// SIMATIC S7-200 project (STEP 7-Micro/WIN), CPU 222 REL 02.01

SYMBOL_TABLE DR03
S1_0300_AdjDigits0 VW1800   // Scale1 - Adjusting digits for zero point
S1_0302_AdjDigits1 VW1802   // Scale1 - Adjusting digits for adjusting weight 1
S1_0304_AdjDigits2 VW1804   // Scale1 - Adjusting digits for adjusting weight 2
S1_0306_AdjWeight1 VW1806   // Scale1 - Adjusting weight 1
S1_0308_AdjWeight2 VW1808   // Scale1 - Adjusting weight 2
S1_0310_CharVal  VB1810   // Scale1 - Characteristic value [mV/V]
S1_0311_MeasuremTime VB1811   // Scale1 - Measurement time, 0=20ms, 1=33,33ms
S1_0312_LimFrequ VB1812   // Scale1 - Limit frequency for low pass filter fg
S1_0313_DepthAvValFiltr VB1813   // Scale1 - Depth of average value filter [0..255]
S1_0314_ScaleName_maxL VB1814   // Scale1 - Scale name, max. length (bytes)
S1_0315_ScaleName_strg VB1815   // Scale1 - Scale name, STRING[10]
S1_0326_MinWeight VW1826   // Scale1 - Minimum weight for weighing range
S1_0328_MaxWeight VW1828   // Scale1 - Maximum weight for weighing range
S1_0330_NumeralStep VW1830   // Scale1 - Numeral step (1, 2, 5, 10, 20)
S1_0332_StandstillRange VW1832   // Scale1 - Standstill range in weight unit
S1_0334_StandstillTime VD1834   // Scale1 - Standstill time in ms
S1_0338_DecimalPoint VB1838   // Scale1 - Decimal place for remote display and       ASCII weight output (0...5)
S1_0339_NegZeroRange VB1839   // Scale1 - Negative range of zero setting device                   [in % of WBB.]
S1_0340_PosZeroRange VB1840   // Scale1 - Positive range of zero setting device                   [in % of WBB.]
S1_0341_TareMax  VB1841   // Scale1 - Subtractive tare device range in % of weighing range
S1_0342_TTYinterface VW1842   // Scale1 - 0: Siebert S102, 1: ASCII protocol
S1_0344_Res_maxL VB1844   // Scale1 - Reserved, max. length (bytes)
S1_0345_Res_strg VB1845   // Scale1 - Reserved, STRING[4]
S1_0350_Unit_maxL VB1850   // Scale1 - Weight unit for display, max. length (bytes)
S1_0351_Unit_strg VB1851   // Scale1 - Weight unit for display, STRING[4]
END_SYMBOL_TABLE

SYMBOL_TABLE DR04
S1_0400_SwOnWeightLim1 VW1856   // Scale1 - Switch on point, limit value 1
S1_0402_SwOffWeightLim1 VW1858   // Scale1 - Switch off point, limit value 1
S1_0404_SwOnWeightLim2 VW1860   // Scale1 - Switch on point, limit value 2
S1_0406_SwOffWeightLim VW1862   // Scale1 - Switch off point, limit value 2
S1_0408_LimValParamFlag VB1864   // Scale1 - Bit0: 0=lim1 on gross, 1=lim1 on net;                Bit1: --> lim2
S1_0409_Res1     VB1865   // Scale1 - Reserve 1
END_SYMBOL_TABLE

SYMBOL_TABLE DR09
S1_0900_ModuleName_maxL VB1866   // Scale1 - Name of weighing module, max. length (bytes)
S1_0901_ModuleName_strg VB1867   // Scale1 - Name of weighing module, STRING[10]
S1_0912_MLFB_maxL VB1878   // Scale1 - MLFB order number, max. length (bytes)
S1_0913_MLFB_strg VB1879   // Scale1 - MLFB order number, STRING[20]
S1_0934_Edition1HW VW1900   // Scale1 - HW version
S1_0936_FWversion_maxL VB1902   // Scale1 - FW version, max. length (bytes)
S1_0937_FWversion_strg VB1903   // Scale1 - FW version, STRING[4]
S1_0942_CRCpackage VW1908   // Scale1 - Depending on code
END_SYMBOL_TABLE

SYMBOL_TABLE MS-Symbols
Command_In_Progress V2004.0  // command in progress
Command_FOK      V2004.1  // command finished ok
Command_ERR      V2004.2  // command error has occurred
Asynchronous_Error_Bit0 V2006.0  // Reboot due to RAM error
Asynchronous_Error_Bit1 V2006.1  // Reboot due to watchdog error
Asynchronous_Error_Bit2 V2006.2  // Power supply faulty/missing
Asynchronous_Error_Bit3 V2006.3  // Number overflow in weight calculation
Asynchronous_Error_Bit4 V2006.4  // Parameter error
Asynchronous_Error_Bit5 V2006.5  // AD converter at limit of measuring range
Asynchronous_Error_Bit6 V2006.6  // Minimum voltage undershot on sensor line
Asynchronous_Error_Bit7 V2006.7  // AD converter fault
Status_write_protection V2008.0  // 1 = Write protect switch active
Status_min_undershot V2008.1  // 1 = Min. weighing range undershot
Status_Bit10     V2008.2  // Reserve
Status_Bit11     V2008.3  // Reserve
Status_Bit12     V2008.4  // Reserve
Status_Bit13     V2008.5  // Reserve
Status_startup   V2008.6  // 1 = startup is running
Status_module_fault V2008.7  // 1 = Global module fault / operating error (SF)
Status_limit1    V2009.0  // 1 = Limit value 1 has responded
Status_limit2    V2009.1  // 1 = Limit value 2 has responded
Status_tare_memory V2009.2  // 1 = Tare memory occupied (<> 0)
Status_tare_preset V2009.3  // 1 = Tare memory contains ext. default value
Status_9_display_steps V2009.4  // 1 = Gross weighing range exceeded or undershot by more than 9 display steps
Status_Gross_less V2009.5  // 1 = Gross less than ± 0.25d (d corresponds to set numeral step)
Status_standstill V2009.6  // 1 = Standstill exists
Status_calibrated V2009.7  // 1 = Module calibrated
Command_Trigger  V2012.0  // Command trigger
Add_Command_trigger V2030.0
Add_Busy         V2030.1
Add_Done         V2030.2
Add_Aborted      V2030.3
Actual_Process_Value VB2000   // actual processvalue (Siwarex => PLC; Value: 0...6)
Bit_Messages     VB2004   // Bit-Messages (Siwarex => PLC)
Synchronous_Error_Code VB2005   // synchronous error code
Asynchronous_Error_Bits VB2006   // asynchronous error (bit by bit)
Refresh_Counter  VB2007   // Refresh counter
Select_Process_Value VB2010   // select processvalue (PLC => Siwarex; Value: 0...6)
Command_Code     VB2011   // Command code
Bit_Commands     VB2012   // Bit-Commands (PLC => Siwarex)
Bit_Saving       VB2013   // internal Bit-saving
RW_Mode_DR_No    VB2020   // libraray internal use
RW_Mode_Byteoffset VB2021   // libraray internal use
Add_Command_Code VB2026
Add_DR           VB2027
Add_Offset       VB2028
Add_Length       VB2029
TD100C_SubroutineBuffer VB2042
Process_Value    VW2002   // PROCESSVALUE (Siwarex => PLC)
Scale_Status_Bits VW2008   // Scale status
Preset_Tare_Value VW2014   // Preset tare value (PLC => Siwarex)
Lifebit_Counter  VW2016   // Lifebit Counter
Lib_Error_Bits   VW2018   // Library Error Bits
RW_Mode_Write_Data VW2022   // libraray internal use
RW_Mode_Read_Data VW2024   // libraray internal use
Add_Error        VW2032
Error_messages1  VW2034   // Error messages for Panel
Error_messages2  VW2036   // Error messages for Panel
Error_messages3  VW2038   // Error messages for Panel
TD100C_Adjustment VW2040   // Adjustment via Panel
END_SYMBOL_TABLE

SYMBOL_TABLE DR15
S1_1500_TareInpVal VW1910   // Scale1 - Tare input value (preset Tare pT)
END_SYMBOL_TABLE

SYMBOL_TABLE DR26
S1_2600_Checksum VW1912   // Scale1 - Checksum
S1_2602_Res      VB1914   // Scale1 - Reserved
S1_2603_PresetTare VB1915   // Scale1 - 1 = Tare memory contains ext. default value
S1_2604_Tare_x100 VD1916   // Scale1 - Tare weight * 100
S1_2608_ZeroSetVal_x100 VD1920   // Scale1 - Zero set value * 100 (set during zero setting)
END_SYMBOL_TABLE

SYMBOL_TABLE DR30
S1_3000_Checksum VW1924   // Scale1 - Checksum CRC16
S1_3002_ScaleStatus VW1926   // Scale1 - Scale status
S1_3004_OpErrorBits VB1928   // Scale1 - Operating error bits
S1_3005_Res1     VB1929   // Scale1 - Reserve 1
S1_3006_GrossProcessVal VW1930   // Scale1 - Gross weight
S1_3008_NetProcessVal VW1932   // Scale1 - Net weight
S1_3010_TareProcessVal VW1934   // Scale1 - Tare weight
S1_3012_GNweight VW1936   // Scale1 - B/N weight value to display
S1_3014_GNweight10 VD1938   // Scale1 - B/N weight value with 10x resolution (basis for ASCII weight value)
S1_3018_TareWeight VW1942   // Scale1 - Tare weight value
S1_3020_UnfiltRawVal VW1944   // Scale1 - Unfiltered digital value from ADU
S1_3022_FiltRawVal VW1946   // Scale1 - Filtered digital value
S1_3024_WghtASCII_maxL VB1948   // Scale1 - ASCII weight value, max. length (bytes)
S1_3025_WghtASCII_strg VB1949   // Scale1 - ASCII weight value, STRING[14]
S1_3040_Millisecond VW1964   // Scale1 - Runtime – Milliseconds (0....999)
S1_3042_Second   VB1966   // Scale1 - Runtime – Seconds (0...59)
S1_3043_Minute   VB1967   // Scale1 - Runtime – Minutes (0...59)
S1_3044_Hour     VW1968   // Scale1 - Runtime – Hours (0...32000)
END_SYMBOL_TABLE

SYMBOL_TABLE S7-200 Symbols
Always_On        SM0.0    // Always ON
END_SYMBOL_TABLE

ORGANIZATION_BLOCK MAIN:OB1
TITLE=
BEGIN
Network 1
// The datablock-size for one SIWAREX MS is 20 Bytes (e.g.: VB0...VB19)
// 
// PARAMETER OF LIBRARY:
// 
// First_AEW:	1. input-word of module address
// Second_AEW:	2. input-word of module address
// Third_AEW:	3. input-word of module address
// Fourth_AEW:	4. input-word of module address
// 
// * * * * * * * * * * * * * * * * * * * * * * * * * * * * * * * * * * * * * * * * * * * * * * * * * * * * * * * * * * * * * * * * 
// *		Note:							   *
// *		The Analog Input Filter must be disabled!			   *
// * * * * * * * * * * * * * * * * * * * * * * * * * * * * * * * * * * * * * * * * * * * * * * * * * * * * * * * * * * * * * * * * 
// 
// FirstVB_POINTER: 	first variable-byte in datablock as POINTER, e.g. "&VB0"
// 		The required length into the Variable memory is 20 Bytes! 
// 
// Lib_Error_Bits:	Bit0...7:    Reserve     
// 		Bit8:          Error in Parameter "FirstVB_POINTER" 
// 		Bit9:          Lifebit-Error Siwarex
//  		Bit10:        Error "select processvalue" (value: 0...6)
//  		Bit11:        Command  not completed caused by startup
// 		Bit12...15: Reserve   
// 
// First_AAW:	1. output-word of module address
// Second_AAW:	2. output-word of module address
// Third_AAW:	3. output-word of module address
// Fourth_AAW:	4. output-word of module address
LD     Always_On:SM0.0
CALL   MicroScale_V20:SBR2, AIW0, AIW2, AIW4, AIW6, &Actual_Process_Value:VB2000, Lib_Error_Bits:VW2018, AQW0, AQW2, AQW4, AQW6
Network 2
LD     Always_On:SM0.0
CALL   MicroScale_additional:SBR1, &Actual_Process_Value:VB2000, &VB1800, Add_Command_Code:VB2026, Add_DR:VB2027, Add_Offset:VB2028, Add_Length:VB2029, Add_Command_trigger:V2030.0, Add_Busy:V2030.1, Add_Done:V2030.2, Add_Aborted:V2030.3, Add_Error:VW2032
Network 3 // TD 100C
LD     Always_On:SM0.0
CALL   TD100C:SBR0, VB2018, Asynchronous_Error_Bits:VB2006, Synchronous_Error_Code:VB2005, Command_ERR:V2004.2, TD_CurScreen_0:VB48, Error_messages1:VW2034, Error_messages2:VW2036, Error_messages3:VW2038, F1:V45.0, F2:V45.1, TD100C_SubroutineBuffer:VB2042, VB2030, Add_Command_Code:VB2026, Add_DR:VB2027, Add_Offset:VB2028, Add_Length:VB2029
END_ORGANIZATION_BLOCK

SUBROUTINE_BLOCK TD100C:SBR0
TITLE=UNTERPROGRAMM-KOMMENTARE
VAR_INPUT
Lib_Error_Bits:BYTE;	// LB0 Library_Error_Bits
Asyn_Error_Bits:BYTE;	// LB1 Asynchronous Error Bits
Syn_Error_Code:BYTE;	// LB2 Synchronous Error Code
Command_ERR:BOOL;	// L3.0 Command Error
PictureNo:BYTE;	// LB4 Picture number
END_VAR
VAR_IN_OUT
Error_Messages1:WORD;	// LW5 Error messages for Panel
Error_Messages2:WORD;	// LW7 Error messages for Panel
Error_Messages3:WORD;	// LW9 Error messages for Panel
F1_Button:BOOL;	// L11.0 Button "F1"
F2_Button:BOOL;	// L11.1 Button "F2"
Subroutine_Buffer:BYTE;	// LB12 internal Subroutine Buffer
Command_Bit_Handling:BYTE;	// LB13 Command Bits (Bit0 = Trigger, Bit1 = Busy)
END_VAR
VAR_OUTPUT
Command_Code:BYTE;	// LB14 Command Code
DR:BYTE;	// LB15 DR-No.
Offset:BYTE;	// LB16 Offset
Lenght:BYTE;	// LB17 Lenght
END_VAR
VAR
Tmp_POINTER:DWORD;	// LD18 temporary Pointer
Tmp_Value:WORD;	// LW22 temporary Scale Status value
END_VAR
BEGIN
Network 1
LD     Always_On:SM0.0
CALL   TD_CTRL_0:SBR3
Network 2 // Command
// Zeroing
//Picture-Nr.
//Command Code
//Command Trigger
// (network saved uncompiled; FBD cells follow)
// row 0: c5 [MOV_B ]
// row 1: c1 [==B #PictureNo:LB4 1 ]  c2 [AND #F1_Button:L11.0 ]  c3 -- v  c4 --  c5 [ EN:=power@row1, IN:=21, ENO=>V?0, OUT=>#Command_Code:LB14]
// row 2: c1 [box]  c2 [box]  c3 ^v  c5 [box]
// row 3: c2 [box]  c3 ^v
// row 4: c3 ^v  c4 --  c5 [S L13.0 N:=1]
// row 5: c3 ^v  c5 [box]
// row 6: c3 ^v
// row 7: c3 ^  c4 --  c5 [R #F1_Button:L11.0 N:=1]
// row 8: c5 [box]
Network 3 // Command
// Tare
//Picture-Nr.
//Command Code
//Command Trigger
// (network saved uncompiled; FBD cells follow)
// row 0: c5 [MOV_B ]
// row 1: c1 [==B #PictureNo:LB4 2 ]  c2 [AND #F1_Button:L11.0 ]  c3 -- v  c4 --  c5 [ EN:=power@row1, IN:=22, ENO=>V?0, OUT=>#Command_Code:LB14]
// row 2: c1 [box]  c2 [box]  c3 ^v  c5 [box]
// row 3: c2 [box]  c3 ^v
// row 4: c3 ^v  c4 --  c5 [S L13.0 N:=1]
// row 5: c3 ^v  c5 [box]
// row 6: c3 ^v
// row 7: c3 ^  c4 --  c5 [R #F1_Button:L11.0 N:=1]
// row 8: c5 [box]
Network 4 // Command
// Delete Tare
//Picture-Nr.
//Command Code
//Command Trigger
// (network saved uncompiled; FBD cells follow)
// row 0: c5 [MOV_B ]
// row 1: c1 [==B #PictureNo:LB4 2 ]  c2 [AND #F2_Button:L11.1 ]  c3 -- v  c4 --  c5 [ EN:=power@row1, IN:=23, ENO=>V?0, OUT=>#Command_Code:LB14]
// row 2: c1 [box]  c2 [box]  c3 ^v  c5 [box]
// row 3: c2 [box]  c3 ^v
// row 4: c3 ^v  c4 --  c5 [S L13.0 N:=1]
// row 5: c3 ^v  c5 [box]
// row 6: c3 ^v
// row 7: c3 ^  c4 --  c5 [R #F2_Button:L11.1 N:=1]
// row 8: c5 [box]
Network 5 // ADJUSTMENT: Read the adjustment weight
LDB=   #PictureNo:LB4, 5
AN     L12.0
=      L12.1                 //edge
LDB=   #PictureNo:LB4, 5
=      L12.0
LD     L12.1                 //edge
S      L12.2, 1
LD     L12.2
AN     L13.0
AN     L13.1
MOVB   3, #DR:LB15           //DR-No.
MOVB   6, #Offset:LB16       //offset = 6 = adjustment weight 1
MOVB   2, #Lenght:LB17       //Lenght
MOVB   254, #Command_Code:LB14 //Read data
S      L13.0, 1              //Command Trigger
R      L12.2, 1
Network 6 // ADJUSTMENT: Write the adjustment weight
//Picture-Nr.
//DR-No.
//offset = 6 = adjustment weight 1
//Lenght
//Write data
//Command Trigger
// (network saved uncompiled; FBD cells follow)
// row 0: c5 [MOV_B ]
// row 1: c1 [==B #PictureNo:LB4 5 ]  c2 [AND #F1_Button:L11.0 ]  c3 -- v  c4 --  c5 [ EN:=power@row1, IN:=3, ENO=>V?0, OUT=>#DR:LB15]
// row 2: c1 [box]  c2 [box]  c3 ^v  c5 [box]
// row 3: c2 [box]  c3 ^v  c5 [MOV_B ]
// row 4: c3 ^v  c4 --  c5 [ EN:=power@row4, IN:=6, ENO=>V?0, OUT=>#Offset:LB16]
// row 5: c3 ^v  c5 [box]
// row 6: c3 ^v  c5 [MOV_B ]
// row 7: c3 ^v  c4 --  c5 [ EN:=power@row7, IN:=2, ENO=>V?0, OUT=>#Lenght:LB17]
// row 8: c3 ^v  c5 [box]
// row 9: c3 ^v  c5 [MOV_B ]
// row 10: c3 ^v  c4 --  c5 [ EN:=power@row10, IN:=255, ENO=>V?0, OUT=>#Command_Code:LB14]
// row 11: c3 ^v  c5 [box]
// row 12: c3 ^v
// row 13: c3 ^v  c4 --  c5 [S L13.0 N:=1]
// row 14: c3 ^v  c5 [box]
// row 15: c3 ^v
// row 16: c3 ^  c4 --  c5 [R #F1_Button:L11.0 N:=1]
// row 17: c5 [box]
Network 7 // ADJUSTMENT: Command "Set as Zero"
// Set as Zero
//Picture-Nr.
//Command Code
//Command Trigger
// (network saved uncompiled; FBD cells follow)
// row 0: c5 [MOV_B ]
// row 1: c1 [==B #PictureNo:LB4 6 ]  c2 [AND #F1_Button:L11.0 ]  c3 -- v  c4 --  c5 [ EN:=power@row1, IN:=3, ENO=>V?0, OUT=>#Command_Code:LB14]
// row 2: c1 [box]  c2 [box]  c3 ^v  c5 [box]
// row 3: c2 [box]  c3 ^v
// row 4: c3 ^v  c4 --  c5 [S L13.0 N:=1]
// row 5: c3 ^v  c5 [box]
// row 6: c3 ^v
// row 7: c3 ^  c4 --  c5 [R #F1_Button:L11.0 N:=1]
// row 8: c5 [box]
Network 8 // ADJUSTMENT: Command "Adjustment weight 1 valid"
// Adjustment weight 1 valid
//Picture-Nr.
//Command Code
//Command Trigger
// (network saved uncompiled; FBD cells follow)
// row 0: c5 [MOV_B ]
// row 1: c1 [==B #PictureNo:LB4 7 ]  c2 [AND #F1_Button:L11.0 ]  c3 -- v  c4 --  c5 [ EN:=power@row1, IN:=4, ENO=>V?0, OUT=>#Command_Code:LB14]
// row 2: c1 [box]  c2 [box]  c3 ^v  c5 [box]
// row 3: c2 [box]  c3 ^v
// row 4: c3 ^v  c4 --  c5 [S L13.0 N:=1]
// row 5: c3 ^v  c5 [box]
// row 6: c3 ^v
// row 7: c3 ^  c4 --  c5 [R #F1_Button:L11.0 N:=1]
// row 8: c5 [box]
Network 9 // error messages
// Delete all alarms
//Picture-Nr.
// (network saved uncompiled; FBD cells follow)
// row 0: c5 [MOV_W ]
// row 1: c1 [==B #PictureNo:LB4 3 ]  c2 [AND #F1_Button:L11.0 ]  c3 -- v  c4 --  c5 [ EN:=power@row1, IN:=0, ENO=>V?0, OUT=>#Error_Messages1:LW5]
// row 2: c1 [box]  c2 [box]  c3 ^v  c5 [box]
// row 3: c2 [box]  c3 ^v  c5 [MOV_W ]
// row 4: c3 ^v  c4 --  c5 [ EN:=power@row4, IN:=0, ENO=>V?0, OUT=>#Error_Messages2:LW7]
// row 5: c3 ^v  c5 [box]
// row 6: c3 ^v  c5 [MOV_W ]
// row 7: c3 ^v  c4 --  c5 [ EN:=power@row7, IN:=0, ENO=>V?0, OUT=>#Error_Messages3:LW9]
// row 8: c3 ^v  c5 [box]
// row 9: c3 ^v
// row 10: c3 ^  c4 --  c5 [R #F1_Button:L11.0 N:=1]
// row 11: c5 [box]
Network 10 // error messages
//The ORB instruction ORs the corresponding bits of two input values
// (network saved uncompiled; FBD cells follow)
// row 0: c4 [WOR_B ]
// row 1: c1 [AND Always_On:SM0.0 ]  c2 -- v  c3 --  c4 [ EN:=power@row1, IN1:=#Lib_Error_Bits:LB0, IN2:=LB5, ENO=>V?0, OUT=>LB5]
// row 2: c2 ^v  c4 [box]
// row 3: c2 ^v  c4 [box]
// row 4: c2 ^v  c4 [WOR_B ]
// row 5: c2 ^  c3 --  c4 [ EN:=power@row5, IN1:=#Asyn_Error_Bits:LB1, IN2:=LB6, ENO=>V?0, OUT=>LB6]
// row 6: c4 [box]
// row 7: c4 [box]
Network 11 // error messages
LDN    #Command_ERR:L3.0
JMP    10
Network 12 // error messages
LDB=   #Syn_Error_Code:LB2, 1
S      L8.0, 1
Network 13 // error messages
LDB=   #Syn_Error_Code:LB2, 2
S      L8.1, 1
Network 14 // error messages
LDB=   #Syn_Error_Code:LB2, 5
S      L8.3, 1
Network 15 // error messages
LDB=   #Syn_Error_Code:LB2, 7
S      L8.4, 1
Network 16 // error messages
LDB=   #Syn_Error_Code:LB2, 8
S      L8.5, 1
Network 17 // error messages
LDB=   #Syn_Error_Code:LB2, 20
S      L8.6, 1
Network 18 // error messages
LDB=   #Syn_Error_Code:LB2, 21
S      L8.7, 1
Network 19 // error messages
LDB=   #Syn_Error_Code:LB2, 77
S      L7.0, 1
Network 20 // error messages
LDB=   #Syn_Error_Code:LB2, 80
S      L7.2, 1
Network 21 // error messages
LDB=   #Syn_Error_Code:LB2, 81
S      L7.3, 1
Network 22 // error messages
LDB=   #Syn_Error_Code:LB2, 82
S      L7.4, 1
Network 23 // error messages
LDB=   #Syn_Error_Code:LB2, 83
S      L7.5, 1
Network 24 // error messages
LDB=   #Syn_Error_Code:LB2, 84
S      L7.6, 1
Network 25 // error messages
LDB=   #Syn_Error_Code:LB2, 85
S      L7.7, 1
Network 26 // error messages
LDB=   #Syn_Error_Code:LB2, 86
S      L10.0, 1
Network 27 // error messages
LDB=   #Syn_Error_Code:LB2, 87
S      L10.1, 1
Network 28 // error messages
LDB=   #Syn_Error_Code:LB2, 88
S      L10.2, 1
Network 29 // error messages
LDB=   #Syn_Error_Code:LB2, 94
S      L10.3, 1
Network 30 // error messages
LDB=   #Syn_Error_Code:LB2, 96
S      L10.4, 1
Network 31 // error messages
LDB=   #Syn_Error_Code:LB2, 100
S      L10.5, 1
Network 32 // error messages
LDB=   #Syn_Error_Code:LB2, 171
S      L10.6, 1
Network 33 // error messages
LDB=   #Syn_Error_Code:LB2, 172
S      L10.7, 1
Network 34 // error messages
LDB=   #Syn_Error_Code:LB2, 173
S      L9.0, 1
Network 35 // error messages
LBL    10
Network 36 // error messages - handling
LD     L6.0
CALL   TD_ALM_0:SBR4, OM001:V39.7
Network 37 // error messages - handling
LD     L6.1
CALL   TD_ALM_0:SBR4, OM002:V39.6
Network 38 // error messages - handling
LD     L6.2
CALL   TD_ALM_0:SBR4, OM022:V39.5
Network 39 // error messages - handling
LD     L6.3
CALL   TD_ALM_0:SBR4, OM007:V39.4
Network 40 // error messages - handling
LD     L6.4
CALL   TD_ALM_0:SBR4, OM005:V39.3
Network 41 // error messages - handling
LD     L6.5
CALL   TD_ALM_0:SBR4, OM017:V39.2
Network 42 // error messages - handling
LD     L6.6
CALL   TD_ALM_0:SBR4, OM018:V39.1
Network 43 // error messages - handling
LD     L6.7
CALL   TD_ALM_0:SBR4, OM019:V39.0
Network 44 // error messages - handling
LD     L5.0
CALL   TD_ALM_0:SBR4, SBR_01:V40.7
Network 45 // error messages - handling
LD     L5.1
CALL   TD_ALM_0:SBR4, SBR_02:V40.6
Network 46 // error messages - handling
LD     L5.2
CALL   TD_ALM_0:SBR4, SBR_03:V40.5
Network 47 // error messages - handling
LD     L5.3
CALL   TD_ALM_0:SBR4, SBR_04:V40.4
Network 48 // error messages - handling
LD     L8.0
CALL   TD_ALM_0:SBR4, CMD001:V40.3
Network 49 // error messages - handling
LD     L8.1
CALL   TD_ALM_0:SBR4, CMD002:V40.2
Network 50 // error messages - handling
LD     L8.3
CALL   TD_ALM_0:SBR4, CMD005:V40.1
Network 51 // error messages - handling
LD     L8.4
CALL   TD_ALM_0:SBR4, CMD007:V40.0
Network 52 // error messages - handling
LD     L8.5
CALL   TD_ALM_0:SBR4, CMD008:V41.7
Network 53 // error messages - handling
LD     L8.6
CALL   TD_ALM_0:SBR4, CMD020:V41.6
Network 54 // error messages - handling
LD     L8.7
CALL   TD_ALM_0:SBR4, CMD021:V41.5
Network 55 // error messages - handling
LD     L7.0
CALL   TD_ALM_0:SBR4, CMD077:V41.4
Network 56 // error messages - handling
LD     L7.2
CALL   TD_ALM_0:SBR4, CMD080:V41.2
Network 57 // error messages - handling
LD     L7.3
CALL   TD_ALM_0:SBR4, CMD081:V41.1
Network 58 // error messages - handling
LD     L7.4
CALL   TD_ALM_0:SBR4, CMD082:V41.0
Network 59 // error messages - handling
LD     L7.5
CALL   TD_ALM_0:SBR4, CMD083:V42.7
Network 60 // error messages - handling
LD     L7.6
CALL   TD_ALM_0:SBR4, CMD084:V42.6
Network 61 // error messages - handling
LD     L7.7
CALL   TD_ALM_0:SBR4, CMD085:V42.5
Network 62 // error messages - handling
LD     L10.0
CALL   TD_ALM_0:SBR4, CMD086:V42.4
Network 63 // error messages - handling
LD     L10.1
CALL   TD_ALM_0:SBR4, CMD087:V42.3
Network 64 // error messages - handling
LD     L10.2
CALL   TD_ALM_0:SBR4, CMD088:V42.2
Network 65 // error messages - handling
LD     L10.3
CALL   TD_ALM_0:SBR4, CMD094:V42.1
Network 66 // error messages - handling
LD     L10.4
CALL   TD_ALM_0:SBR4, CMD096:V42.0
Network 67 // error messages - handling
LD     L10.5
CALL   TD_ALM_0:SBR4, CMD100:V43.7
Network 68 // error messages - handling
LD     L10.6
CALL   TD_ALM_0:SBR4, CMD171:V43.6
Network 69 // error messages - handling
LD     L10.7
CALL   TD_ALM_0:SBR4, CMD172:V43.5
Network 70 // error messages - handling
LD     L9.0
CALL   TD_ALM_0:SBR4, CMD173:V43.4
END_SUBROUTINE_BLOCK

// SBR1: protected block, not included

// SBR2: protected block, not included

// SBR3: protected block, not included

// SBR4: protected block, not included

// (further data pages could not be read)
